FUNCTION getTaskCycleTime : UDINT  // return cycle time in integer multiples of 100 ns
VAR_INPUT
END_VAR
VAR
END_VAR

getTaskCycleTime := TwinCAT_SystemInfoVarList._TaskInfo[GETCURTASKINDEXEX()].CycleTime;

END_FUNCTION

(* stored: Version 1.1.0.1, ProductVersion 3.1.4024.15
   POU getTaskCycleTime: Id {8d867274-71e4-4630-a343-5a60566d8a1b}, SpecialFunc None *)
